FUNCTION_BLOCK a1 (* Basic FB with empty ECC *)
  (* Standard: 61499-2 *)
  (* Version 1.0, 2025-03-31, 06220625900 *)
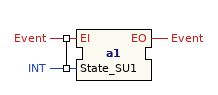
  EVENT_INPUT
    EI WITH State_SU1;
  END_EVENT
  EVENT_OUTPUT
    EO;
  END_EVENT
  VAR_INPUT
    State_SU1 : INT := 1;
  END_VAR
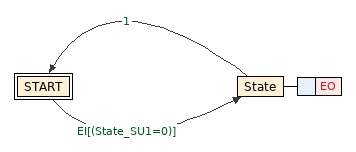
  EC_STATES
    START; (* Initial State *)
    State : -> EO;
  END_STATES
  EC_TRANSITIONS
    START TO State := EI[(State_SU1=0)];
    State TO START := 1;
  END_TRANSITIONS
END_FUNCTION_BLOCK
